PROGRAM PRG_Flow


VAR

i : INT;;

    END_VAR

END_PROGRAM

END_PROGRAM


    //单个功能验证测试


 Act_Manual ();


    //流程寸进


 Act_Step ();


    //流程空跑


 Act_FlowTest ();


    //自动流程


 Act_Auto ();

ACTION Act_Auto:
(*自动控制流程中—>需要用到的控制参数尽量在哪里用就在那里复位清除*)

END_PROGRAM
END_ACTION

ACTION Act_FlowTest:
END_PROGRAM

    // 上使能


    //FOR i:=1 TO iAxisMaxNum BY 1 DO
 

    //	afbAxis[i].xPowerEn := TRUE;
 

    //	afbAxis[i].xPosDirEn := TRUE;
 

    //	afbAxis[i].xNegDirEn := TRUE;
 

    //	afbAxis[i].lrOverride := 100;
 

    //END_FOR
END_ACTION

ACTION Act_Manual:

END_ACTION

ACTION Act_Step:

END_ACTION

END_PROGRAM

(* stored: Version 1.1.0.1, ProductVersion 3.1.4024.12
   POU PRG_Flow: Id {62474feb-6d0c-4d83-8ea1-1897b651e856}, SpecialFunc None
   Action Act_Auto: Id {e378297c-517d-429c-9080-6c35707e882b}
   Action Act_FlowTest: Id {faba86e8-2cba-4e76-af39-3e78e0fc3640}
   Action Act_Manual: Id {87e6a905-5ee0-46f6-b682-fa61e0c45827}
   Action Act_Step: Id {afe1f34b-674e-48d4-8d68-833b91b590f7} *)
